// SIMATIC S7-200 project (STEP 7-Micro/WIN), CPU 221 REL 01.10

SYMBOL_TABLE USUARIO1
Q1               I0.0     // Guardamotores en serie de motores (NA)
PG               I0.1     // Pulsador de paro (NC)
PM               I0.2     // Pulsador de marcha
B1               I0.3     // Barrera fotoeléctrica detección cajas.
B2               I0.4     // Barrera fotoeléctrica detección bolsas.
M1               Q0.0     // Cinta transportadora 1.
M2               Q0.1     // Cinta transportadora 2.
H1               Q0.2     // Señalización falla de algún motor
H2               Q0.3     // Señalización de proceso en marcha.
END_SYMBOL_TABLE

ORGANIZATION_BLOCK PRINCIPAL:OB1
TITLE=COMENTARIOS DEL PROGRAMA
BEGIN
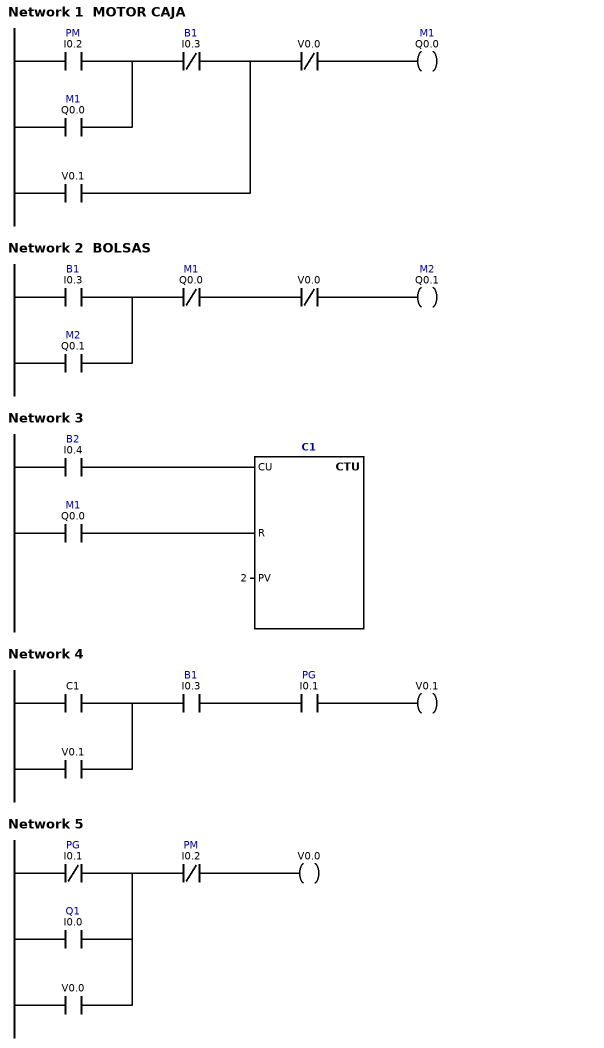
Network 1 // MOTOR CAJA
LD     PM:I0.2
O      M1:Q0.0
AN     B1:I0.3
O      V0.1
AN     V0.0
=      M1:Q0.0
Network 2 // BOLSAS
LD     B1:I0.3
O      M2:Q0.1
AN     M1:Q0.0
AN     V0.0
=      M2:Q0.1
Network 3
LD     B2:I0.4
LD     M1:Q0.0
CTU    C1, 2
Network 4
LD     C1
O      V0.1
A      B1:I0.3
A      PG:I0.1
=      V0.1
Network 5
LDN    PG:I0.1
O      Q1:I0.0
O      V0.0
AN     PM:I0.2
=      V0.0
END_ORGANIZATION_BLOCK
